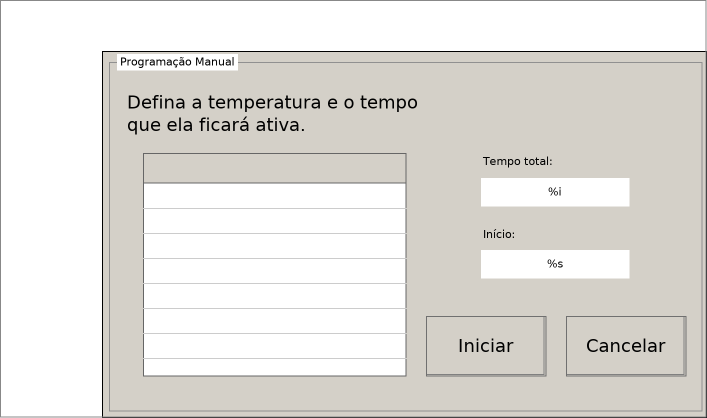
VISUALIZATION TimeCustom_2  // 707x418
    Rectangle (102,51 605x367)
    GroupBox (109,54 593x357), "Programação Manual"
        Button (457,262 120x60), "Cancelar"
            OnMouseClick: CloseDialog Dialog=TimeCustom_2, Result=OK, NumpadKeypadSet=True
        Button (317,262 120x60), "Iniciar"
            OnMouseClick: CloseDialog Dialog=TimeCustom_2, Result=OK, NumpadKeypadSet=True
            OnMouseClick: execute { simIniciaProg_Manual_2(); }
        Label (371,96 73x23), "Tempo total:"
        Textfield (371,123 150x30), "%i", text variable: GVL.totalManual[1]
    Table (143,153 263x223), data array: GVL_P.arr_CustomTime_020
        p3854506369: GVL_P.arr_CustomTime_020[0,INDEX]
        p1892666644: GVL_P.arr_CustomTime_020[1,INDEX]
        p2232123230: TEMPERATURA (ºC)
        p511219082: TEMPO (H)
        Columns.Column.[0].Template: OnMouseUp: write the text variable via VisuDialogs.Numpad
        Columns.Column.[1].Template: OnMouseUp: write the text variable via VisuDialogs.Numpad
    Label (124,90 305x50), "Defina a temperatura e o tempo que ela ficará ativa."
    Textfield (480,249 150x30), "%s", text variable: GVL.progInicio[GVL.actEst]
        OnMouseClick: OpenDialog Dialog=setInicio, OpenModal=True, OpenCentered=True
        OnMouseClick: execute {
            gvl.dia:= MID(STR:= gvl.progInicio[gvl.actEst] , LEN:= 2, POS:=12);
            gvl.mes:= MID(STR:= gvl.progInicio[gvl.actEst] , LEN:= 2, POS:=9);
            gvl.ano:= MID(STR:= gvl.progInicio[gvl.actEst] , LEN:= 2, POS:=6);
            gvl.hora:= MID(STR:= gvl.progInicio[gvl.actEst] , LEN:= 2, POS:=15);
            gvl.minuto:= MID(STR:= gvl.progInicio[gvl.actEst] , LEN:= 2, POS:=18);
        }
    Label (480,223 57x23), "Início:"
END_VISUALIZATION

(* stored: Version 1.1.0.1, ProductVersion 3.1.4024.12
   Visu TimeCustom_2: Id {ddfe0356-2edb-4002-89a9-175c3487de3b} *)
